TYPE INTERNAL ST_BroadcastObject :
STRUCT
	iObj		: U_BroadcastObject;
	nType		: USINT;
END_STRUCT
END_TYPE

(* stored: Version 1.1.0.1
   DUT ST_BroadcastObject: Id {c7a7d29f-efe7-4297-b94b-aa4eb559cb25} *)
